# EPICS autosave request: iocBoot/ioc1/dbSave/KB_Vy_.req
%
% BURT Request File
%
% $(P)KB:Vy:  Vertical KB mirror Y-positioning
%

file assy.req ASSY=$(P)KB:Vy
$(P)KB:Vy:BaseLength
file mtr1.req MTR1=$(P)KB:mvy1
file mtr1.req MTR1=$(P)KB:mvy2
file drv1.req DRV1=$(P)KB:VY1
file drv1.req DRV1=$(P)KB:VY2
file axs1.req AXS1=$(P)KB:VL
file axs1.req AXS1=$(P)KB:VW
